{attribute 'GeneratedUsingTerminal: EL3773-0000-0018'}
{attribute addProperty BoxType "EL3773-0000-0018"}
{attribute addProperty Id "U2_StatusAT %I*U2_Status_DC9039207"}
{attribute addProperty CRC "219681790"}
{attribute addProperty Size "7"}
TYPE L2_Voltage_Status_0D1813FE EXTENDS InputBase_8311D824 :
STRUCT
	{attribute addProperty Name "U2_Status"}
	U2_Status AT %I* : U2_Status_DC903920;
END_STRUCT
END_TYPE

(* stored: Version 1.2.0.0, ProductVersion 3.1.4024.11
   DUT L2_Voltage_Status_0D1813FE: Id {1e3e4d45-b1fa-43d5-b571-27e2885c31ac} *)
